(* IEC 61131-3 sources: axftcmlib/test/Motion/commands, 4 files *)

(* ---- dummy.st ---- *)
USING AxUnit.Assert;
USING Simatic.Ax.Commands;
USING Simatic.Ax.SimpleControlModules;

NAMESPACE Simatic.Ax.axftcmlib.Motion

    {TestFixture}
    CLASS dummy
        VAR

        END_VAR

        {TestSetup}
        METHOD PUBLIC TestSetup
            ;
        END_METHOD

        {Test}
        METHOD PUBLIC TestMethod
            ;
        END_METHOD
    END_CLASS
END_NAMESPACE

(* ---- testCommandActiveHoming.st ---- *)
USING Simatic.Ax.IO.Input;
USING AxUnit.Assert;
USING Simatic.Ax.Commands;
USING Simatic.Ax.SimpleControlModules;

NAMESPACE Simatic.Ax.axftcmlib.Motion

    {TestFixture}
    CLASS testCommandActiveHoming
        VAR
            axis : PosAxis;
            axisStateLess : PosAxis;
            toAxis : TO_PosAxis;
            toAxisStateLess : TO_PosAxis;
            command : itfCommand;
            cmdHomeDirect : commandActiveHoming;
            encoder : MockEncoder;
            RefSensor : BinSignal;
            M1 : MotorBiDirectional;
        END_VAR

        {TestSetup}
        METHOD PUBLIC TestSetup
            axis := axisStateLess;
            toAxis := toAxisStateLess;
            toAxis.Encoder := encoder;
            toAxis.Motor := M1;
            ;
        END_METHOD

        {Test}
        METHOD PUBLIC Start_Homing_And_IS_Running_On
            axis.Attach(REF(toAxis));
            axis.PowerOn();
            command := cmdHomeDirect.Start(AxisRef := REF(toAxis), Position := 100.0, RefSensor := RefSensor);
            IF (command <> NULL) THEN
                Equal(expected := TRUE, actual := command.Busy());
                ;
            END_IF;
            Equal(expected := TRUE, actual := toAxis.IsRunning());

            // set the encoder position manually to 100
            encoder.SetValue(100);

            Equal(expected := FALSE, actual := command.Done());
            Equal(expected := TRUE, actual := toAxis.IsRunning());

            RefSensor.ReadCyclic(signal := TRUE);
            Equal(expected := TRUE, actual := command.Done());
            Equal(expected := FALSE, actual := toAxis.IsRunning());
            Equal(expected := 100.0, actual := toAxis.GetPosition());

        END_METHOD
    END_CLASS

END_NAMESPACE

(* ---- testCommandHome.st ---- *)
USING AxUnit.Assert;
USING Simatic.Ax.Commands;
USING Simatic.Ax.SimpleControlModules;

NAMESPACE Simatic.Ax.axftcmlib.Motion

    {TestFixture}
    CLASS testCommandHome
        VAR
            axis : PosAxis;
            axisStateLess : PosAxis;
            toAxis : TO_PosAxis;
            toAxisStateLess : TO_PosAxis;
            command : itfCommand;
            cmdHomeDirect : commandHomeDirect;
            encoder : MockEncoder;
        END_VAR

        {TestSetup}
        METHOD PUBLIC TestSetup
            axis := axisStateLess;
            toAxis := toAxisStateLess;
            toAxis.Encoder := encoder;
            ;
        END_METHOD

        {Test}
        METHOD PUBLIC CommandHome_To_100_Set_Position_to_100
            axis.Attach(REF(toAxis));
            axis.PowerOn();
            command := cmdHomeDirect.Start(AxisRef := REF(toAxis), Position := 100.0);
            Equal(expected := 100.0, actual := toAxis.GetPosition());
        END_METHOD
        {Test}
        METHOD PUBLIC An_running_Axis_cant_be_homed
            axis.Attach(REF(toAxis));
            axis.PowerOn();
            axis.MoveVelocity(100.0, Direction#PositiveDirection);
            command := cmdHomeDirect.Start(AxisRef := REF(toAxis), Position := 100.0);
            Equal(expected := TRUE, actual := command.Error());
            NotEqual(expected := WORD#0000, actual := command.ErrorID());
            Equal(expected := 0.0, actual := toAxis.GetPosition());
        END_METHOD
    END_CLASS

    CLASS MockEncoder IMPLEMENTS IEncoder
        VAR PUBLIC

        END_VAR
        VAR PROTECTED
            _value : LINT;
        END_VAR

        METHOD PUBLIC MyMethod
            ;
        END_METHOD

        METHOD PUBLIC Evaluate
            ;
        END_METHOD

        METHOD PUBLIC Reset
            ;
        END_METHOD

        METHOD PUBLIC SetValue
            VAR_INPUT
                value : LINT;
            END_VAR
            _value := value;
            ;
        END_METHOD

        METHOD PUBLIC GetValue : LINT
            GetValue := _value;
        END_METHOD

        METHOD PUBLIC SetDirection
            VAR_INPUT
                mode : CountMode;
            END_VAR

            ;
        END_METHOD

        METHOD PUBLIC RelativeCount : LINT
            ;
        END_METHOD

        METHOD PUBLIC ResetRelative
            ;
        END_METHOD

        METHOD PUBLIC GetModulo : LINT
            ;
        END_METHOD
    END_CLASS

END_NAMESPACE

(* ---- testMoveRelative.st ---- *)
USING AxUnit.Assert;
USING Simatic.Ax.Commands;
USING Simatic.Ax.SimpleControlModules;

NAMESPACE Simatic.Ax.axftcmlib.Motion

    {TestFixture}
    CLASS testMoveRelative
        VAR
            to_pos : TO_PosAxis;
            to_pos_Stateless : TO_PosAxis;
            moveRelative : commandMoveRelative;
            moveRelativeStateLess : commandMoveRelative;
            cmd : itfCommand;
            encoder : MockEncoder;
            motor : MotorFT;
        END_VAR

        {TestSetup}
        METHOD PUBLIC TestSetup
            to_pos := to_pos_Stateless;
            moveRelative := moveRelativeStateLess;
            to_pos.Motor := motor;
            to_pos.Encoder := encoder;
        END_METHOD

        {Test}
        METHOD PUBLIC Start_not_homed_axis_returns_error
            to_pos.isPowerdOn := TRUE;
            cmd := moveRelative.Start(AxisRef := REF(to_pos));
            Equal(expected := TRUE, actual := cmd.Error());
            Equal(expected := WORD#16#8003, actual := cmd.ErrorID());
            to_pos.SetPosition(0);
            cmd := moveRelative.Start(AxisRef := REF(to_pos), distance := 100);
            // Equal(expected := TRUE, actual := cmd.Busy());
            ;
        END_METHOD

        // {Test}
        // METHOD PUBLIC Start_Homed_Axis_with_Distance_100_returns_busy
            // to_pos.isPowerdOn := TRUE;
            // to_pos.SetPosition(0);
            // cmd := moveRelative.Start(AxisRef := REF(to_pos), distance := 100);
            // Equal(expected := TRUE, actual := cmd.Busy());
            // Equal(expected := TRUE, actual := to_pos.IsRunning());
            // encoder.SetValue(100);
            // Equal(expected := TRUE, actual := cmd.Done());
            // Equal(expected := FALSE, actual := to_pos.IsRunning());
            // ;
        // END_METHOD
    END_CLASS
END_NAMESPACE
